// SIMATIC S7-200 project (STEP 7-Micro/WIN), CPU 224 REL 02.01

SYMBOL_TABLE USUARIO1
PULSADOR         I0.0
FC_SUBIDA        I0.1
FC_BAJADA        I0.2
SUBIDA           Q0.0
BAJADA           Q0.1
END_SYMBOL_TABLE

ORGANIZATION_BLOCK PRINCIPAL:OB1
TITLE=COMENTARIOS DEL PROGRAMA
BEGIN
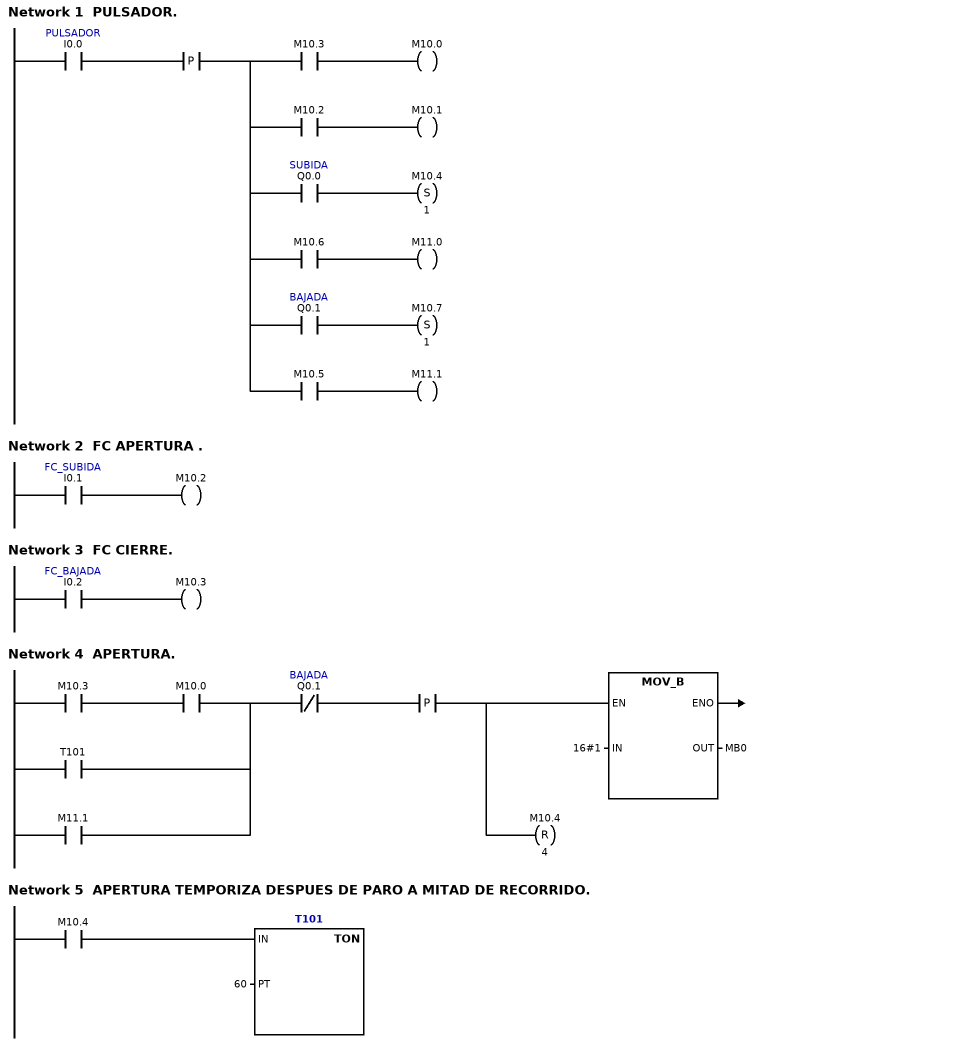
Network 1 // PULSADOR.
LD     PULSADOR:I0.0
EU
LPS
A      M10.3
=      M10.0
LRD
A      M10.2
=      M10.1
LRD
A      SUBIDA:Q0.0
S      M10.4, 1
LRD
A      M10.6
=      M11.0
LRD
A      BAJADA:Q0.1
S      M10.7, 1
LPP
A      M10.5
=      M11.1
Network 2 // FC APERTURA .
LD     FC_SUBIDA:I0.1
=      M10.2
Network 3 // FC CIERRE.
LD     FC_BAJADA:I0.2
=      M10.3
Network 4 // APERTURA.
LD     M10.3
A      M10.0
O      T101
O      M11.1
AN     BAJADA:Q0.1
EU
MOVB   16#1, MB0
R      M10.4, 4
Network 5 // APERTURA TEMPORIZA DESPUES DE PARO A MITAD DE RECORRIDO.
LD     M10.4
TON    T101, 60
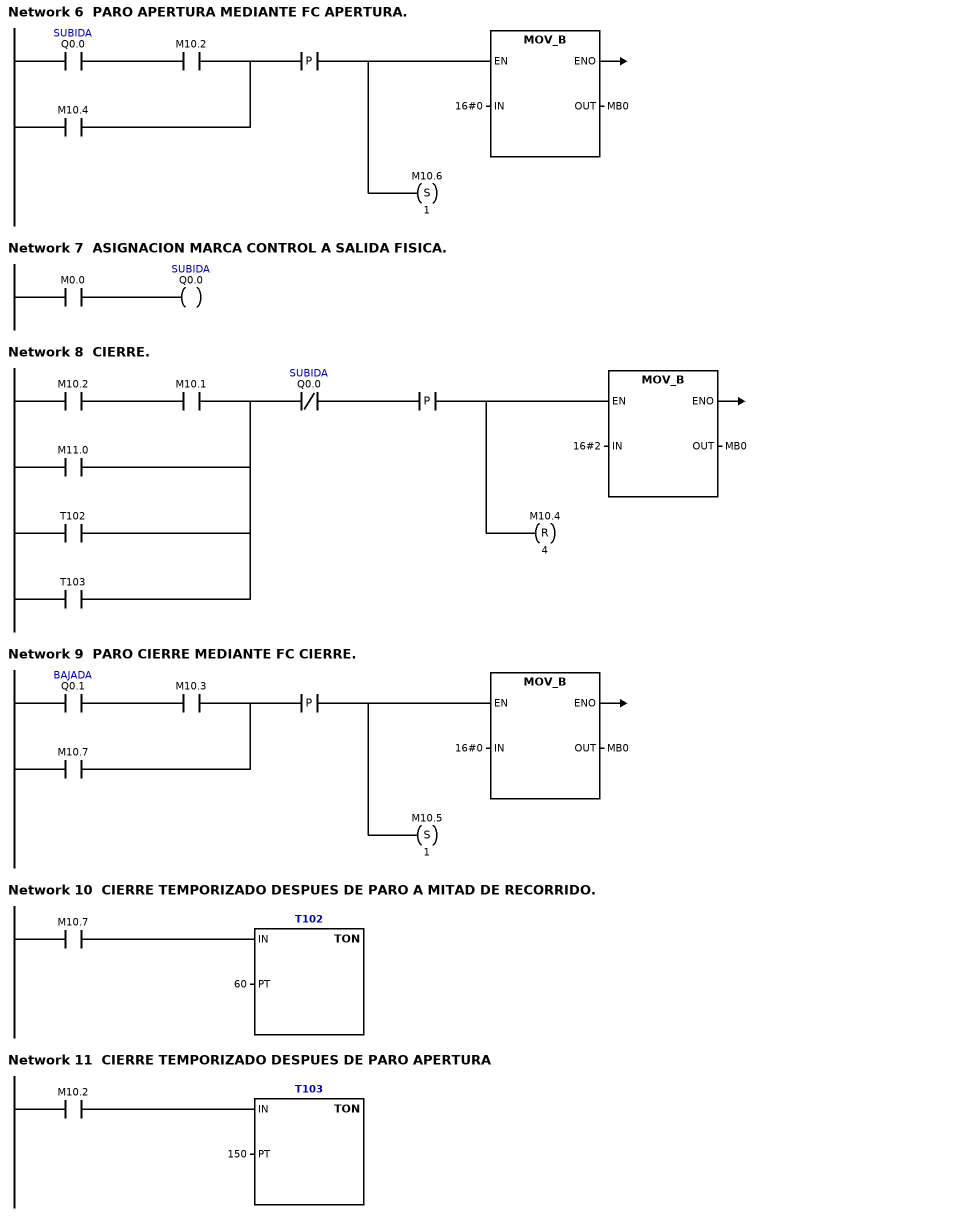
Network 6 // PARO APERTURA MEDIANTE FC APERTURA.
// (network saved uncompiled; LAD cells follow)
// row 0: c0 -| |- SUBIDA:Q0.0  c1 -| |- M10.2 v  c2 -|P|-  v  c3 --  c4 [MOV_B EN:=power@row0, IN:=16#0, ENO=>power, OUT=>MB0]  c5 ->
// row 1: c0 -| |- M10.4  c1 -- ^  c2 ^v  c4 [box]
// row 2: c2 ^  c3 -(S) M10.6, 1
Network 7 // ASIGNACION MARCA CONTROL A SALIDA FISICA.
// (network saved uncompiled; LAD cells follow)
// row 0: c0 -| |- M0.0  c1 -( ) SUBIDA:Q0.0
Network 8 // CIERRE.
// (network saved uncompiled; LAD cells follow)
// row 0: c0 -| |- M10.2  c1 -| |- M10.1 v  c2 -|/|- SUBIDA:Q0.0  c3 -|P|-  v  c4 --  c5 [MOV_B EN:=power@row0, IN:=16#2, ENO=>power, OUT=>MB0]  c6 ->
// row 1: c0 -| |- M11.0  c1 -- ^v  c3 ^v  c5 [box]
// row 2: c0 -| |- T102  c1 -- ^v  c3 ^  c4 -(R) M10.4, 4
// row 3: c0 -| |- T103  c1 -- ^
Network 9 // PARO CIERRE MEDIANTE FC CIERRE.
LD     BAJADA:Q0.1
A      M10.3
O      M10.7
EU
MOVB   16#0, MB0
S      M10.5, 1
Network 10 // CIERRE TEMPORIZADO DESPUES DE PARO A MITAD DE RECORRIDO.
// (network saved uncompiled; LAD cells follow)
// row 0: c0 -| |- M10.7  c1 --  c2 [TON T102 IN:=power@row0, PT:=60]
// row 1: c2 [box]
Network 11 // CIERRE TEMPORIZADO DESPUES DE PARO APERTURA 
LD     M10.2
TON    T103, 150
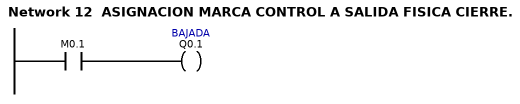
Network 12 // ASIGNACION MARCA CONTROL A SALIDA FISICA CIERRE.
// (network saved uncompiled; LAD cells follow)
// row 0: c0 -| |- M0.1  c1 -( ) BAJADA:Q0.1
END_ORGANIZATION_BLOCK
